Fanuc KAREL source: kd00028.KL

-- PROVISIONAL review KL for V940-1; original PC SHA256 dcd7fc477baadff422aa940cf943a3a662447ed58739e590b315561ed47f03ee
-- Incomplete behavior may be omitted. Consult companion uncertainty JSON. Do not deploy.
PROGRAM KD00028
%NOLOCKGROUP
VAR
  I : INTEGER
  J : INTEGER
  B : BOOLEAN
  R : REAL
  S : STRING[80]
BEGIN
  -- V9_ZERO_TABLE_METADATA_HINT layout=0001; no indexed target words; source/name/runtime held
  -- UNRESOLVED_PC offsets 5-21; opcodes 9D,81,18,9D,12,22,9D,13,04
  -- UNRESOLVED_PC offsets 26-30; opcodes 7F
END KD00028
